FUNCTION_BLOCK fb_ac_ratio_ctrl

VAR_INPUT
	(*
	set_ya:  REAL := g_set_ya;
	set_yac: REAL := g_set_yac;
	xmeas11: REAL := g_xmeas[11];
	xmeas23: REAL := g_xmeas[23];
	xmeas25: REAL := g_xmeas[25];
	*)
END_VAR

VAR_OUTPUT
END_VAR

VAR
	// A & C measurements
	yA: 	REAL;
	yAC:	REAL;
	
	// yA control looop
	ya_control: fb_vel_pi := (kc := 0.0002, ti := 1.0, ts := g_Ts);
	ya_control_kc :	REAL := 0.0;
	loop14:	REAL := 0.0;
	
	// yAC control loop
	yac_control: fb_vel_pi := (kc := 0.0003, ti := 2, ts := g_Ts);
	loop15: REAL := 0.0;	
	
	// ratio trimming
	ratio_trimming: fb_ratio_trimming;
	
	// fine ac adjustments
	ac_measurements: fb_ac_measurements;
	separator_temp_dpi: fb_discrete_pi		:= (kc:=-4, ti:=15/60, Ts:=g_Ts_base, hi :=100, lo:=0, yout:=xmv_0[11]);	
	ratio_trimming_0: fb_ratio_trimming 	:= (r1 := g_rx[1], r4 := g_rx[4]);

END_VAR

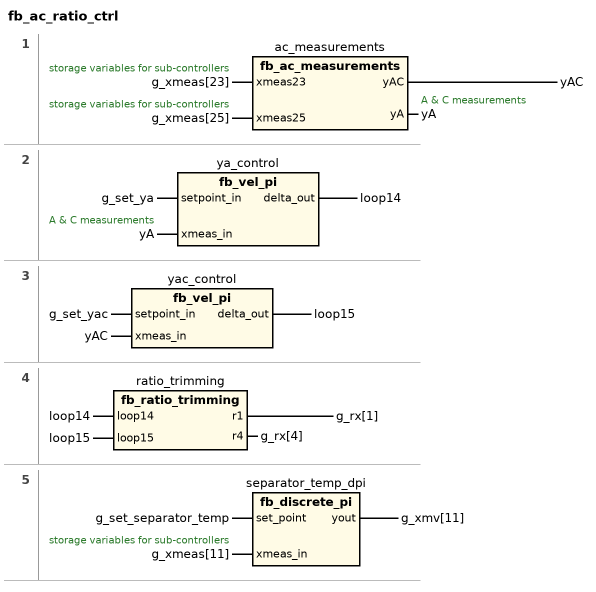
// NETWORK 1
//   ac_measurements: fine ac adjustments
//   g_xmeas[23]: storage variables for sub-controllers
//   g_xmeas[25]: storage variables for sub-controllers
//   yA: A & C measurements
ac_measurements(xmeas23 := g_xmeas[23], xmeas25 := g_xmeas[25], yA => yA); // fb_ac_measurements
yAC := ac_measurements.yAC;

// NETWORK 2
//   ya_control: yA control looop
//   yA: A & C measurements
ya_control(setpoint_in := g_set_ya, xmeas_in := yA); // fb_vel_pi
loop14 := ya_control.delta_out;

// NETWORK 3
//   yac_control: yAC control loop
yac_control(setpoint_in := g_set_yac, xmeas_in := yAC); // fb_vel_pi
loop15 := yac_control.delta_out;

// NETWORK 4
//   ratio_trimming: ratio trimming
ratio_trimming(loop14 := loop14, loop15 := loop15, r4 => g_rx[4]); // fb_ratio_trimming
g_rx[1] := ratio_trimming.r1;

// NETWORK 5
//   g_xmeas[11]: storage variables for sub-controllers
separator_temp_dpi(set_point := g_set_separator_temp, xmeas_in := g_xmeas[11]); // fb_discrete_pi
g_xmv[11] := separator_temp_dpi.yout;

END_FUNCTION_BLOCK

(* stored: Version 1.1.0.1, ProductVersion 3.1.0.26
   POU fb_ac_ratio_ctrl: Id {86afd01c-b43a-4f54-91b7-7c37e6d453f0} *)
